TYPE ST_Instrument :
STRUCT
	
m_armId:INT;
m_instruNameCH : WSTRING;
m_instrumentSN:ULINT;
m_instruUsageCounts :ULINT;
m_maxUseNum :UINT;

END_STRUCT
END_TYPE

(* stored: Version 1.1.0.1, ProductVersion 3.1.4024.11
   DUT ST_Instrument: Id {d2ec0342-e6f0-4f42-8b66-5c50f7d89450} *)
